{attribute 'linkalways'} 
{attribute 'no_explicit_call' := 'This FB is a CLASS and must be accessed using methods or properties'}
{attribute 'enable_dynamic_creation'}
FUNCTION_BLOCK _Array0to1OfUSINT EXTENDS ArrayDatatypeBase_1D
VAR CONSTANT
	lBound : DINT := 0;
	uBound : DINT := 1;
END_VAR
VAR
	localData : ARRAY [lBound..uBound] OF USINT;
	activeData : REFERENCE TO ARRAY [lBound..uBound] OF USINT REF= localData;
	elements : ARRAY [lBound..uBound] OF _USINT(0);
	baseType : _USINT(0);
END_VAR

PROPERTY PUBLIC Address : PVOID
GET
Address := ADR(activeData);
END_GET
END_PROPERTY

PROPERTY PUBLIC BaseDatatype : I_Datatype
GET
BaseDatatype := baseType;
END_GET
END_PROPERTY

METHOD PUBLIC ClearReference
VAR_INPUT
END_VAR
activeData REF= localData;
SetElementReference();
END_METHOD

METHOD PUBLIC Clone : I_Datatype
VAR
    pClone : POINTER TO _Array0to1OfUSINT;
END_VAR
pClone := __NEW(_Array0to1OfUSINT());
pClone^.Value := Value;
Clone := pClone^;
END_METHOD

METHOD FB_init : BOOL
VAR_INPUT
	bInitRetains : BOOL; // if TRUE, the retain variables are initialized (warm start / cold start)
	bInCopyCode : BOOL;  // if TRUE, the instance afterwards gets moved into the copy code (online change)
END_VAR
SetElementReference();
END_METHOD

METHOD PUBLIC MakeReferenceTo
VAR_INPUT
	ReferenceTarget : REFERENCE TO ARRAY [lBound..uBound] OF USINT;
END_VAR
activeData REF= ReferenceTarget;
SetElementReference();
END_METHOD

METHOD PROTECTED OnSerializeArrayValues
VAR_INPUT
	Serializer : I_Serializer;
END_VAR
VAR
	i : DINT;
END_VAR
FOR i := lBound TO uBound DO
	elements[i].SerializeWith(Serializer);
END_FOR
END_METHOD

METHOD PROTECTED SetElementReference
VAR_INPUT
END_VAR
VAR
	i : DINT;
END_VAR
FOR i := lBound TO uBound DO
	elements[i].MakeReferenceTo(activeData[i]);
END_FOR
END_METHOD

PROPERTY PUBLIC Size : UDINT
GET
Size := SIZEOF(activeData);
END_GET
END_PROPERTY

METHOD PROTECTED TryDeserializeArrayValues : BOOL
VAR_INPUT
	Deserializer : I_Deserializer;
	Feedback : I_DeserializerFeedback;
END_VAR
VAR
	enumerator : I_DeserializerArrayForwardEnumerator;
	i : DINT;
END_VAR
enumerator := Deserializer.GetArrayEnumerator();
i := lBound;

WHILE enumerator.MoveNext() AND i <= uBound DO
	
	IF NOT elements[i].TryDeserializeFrom(enumerator.Current, Feedback) THEN
		EXIT;
	END_IF
	i := i + 1;

END_WHILE
enumerator.Dispose();
END_METHOD

METHOD PUBLIC TryGetElementAsDatatypeByIndex : BOOL
VAR_INPUT
	Index : DINT;
	Destination : REFERENCE TO I_Datatype;
END_VAR
IF Index < lbound OR Index > ubound THEN
	RETURN;
END_IF

Destination := elements[Index];
TryGetElementAsDatatypeByIndex := TRUE;
END_METHOD

METHOD PUBLIC TryGetLowerBound : BOOL
VAR_INPUT
	Dimention : UDINT;
	Destination : REFERENCE TO DINT;
END_VAR
IF Dimention = 1 THEN
	Destination := lBound;
	TryGetLowerBound := TRUE;
END_IF
END_METHOD

METHOD PUBLIC TryGetUpperBound : BOOL
VAR_INPUT
	Dimention : UDINT;
	Destination : REFERENCE TO DINT;
END_VAR
IF Dimention = 1 THEN
	Destination := uBound;
	TryGetUpperBound := TRUE;
END_IF
END_METHOD

METHOD TryMakeReferenceTo : BOOL
VAR_INPUT
	Target : I_Datatype;
END_VAR
VAR
	pTargetData : POINTER TO ARRAY [lBound..uBound] OF USINT;
END_VAR
IF NOT IsEquivalentTo(Target) THEN
	RETURN;
END_IF

pTargetData := Target.Address;
activeData REF= pTargetData^;
SetElementReference();
TryMakeReferenceTo := TRUE;
END_METHOD

PROPERTY PUBLIC Value : REFERENCE TO ARRAY [lBound..uBound] OF USINT;
GET
Value ref= activeData;
END_GET
END_PROPERTY

END_FUNCTION_BLOCK

(* stored: Version 1.1.0.1, ProductVersion 3.1.4024.13
   POU _Array0to1OfUSINT: Id {809f4d15-75a6-0d4d-342f-d4df08bef26b}, SpecialFunc None
   Folder Core: Id {20405364-43c1-0360-3f13-c7b6b46347e7}
   Folder Constructor: Id {908c995d-d65e-0f17-2c61-dd1428a238a9}
   Folder Protected: Id {dfab63e4-fcbe-0bc7-0ff3-1ff4a2700262}
   Folder Customize: Id {9282016e-9e25-0a51-3ea2-b0f729feb462}
   Property Address: Id {ad213f99-3e13-0541-3bbf-09cab285d405}
   Get Get: Id {3ed5b802-24ab-0f0e-0445-8231e37b8cbd}
   Property BaseDatatype: Id {7ef03571-8bc5-0247-333b-5691cc5bf9a1}
   Get Get: Id {de10912a-e5a7-03eb-05d8-57eb7747a96a}
   Method ClearReference: Id {ce4594e1-2b13-0cda-2807-59ba5d9189e5}
   Method Clone: Id {64423a02-b6d0-0e8a-0760-8bfc10b30d4b}
   Method FB_init: Id {406c2806-71c0-00af-1989-a14c1a329468}
   Method MakeReferenceTo: Id {5b4f1f2e-542e-0474-1042-eaa2ddcf0ffe}
   Method OnSerializeArrayValues: Id {b21bb398-199d-0e16-31a8-cd09df871397}
   Method SetElementReference: Id {7c9dd691-accb-0531-2dc9-c10ab7ee6fcb}
   Property Size: Id {49787b77-9a41-0c14-15da-d9010493de80}
   Get Get: Id {5634b85b-70c4-0de8-2a44-a0a05d06768a}
   Method TryDeserializeArrayValues: Id {02d736b4-f63d-0bf4-14f9-cfb9fc342882}
   Method TryGetElementAsDatatypeByIndex: Id {32fcd423-74eb-05b7-378c-6b6a234ace87}
   Method TryGetLowerBound: Id {cbf098bf-2dc2-04a7-3516-030d4bd95e11}
   Method TryGetUpperBound: Id {6d144c83-c8ac-0241-2669-af811d77153e}
   Method TryMakeReferenceTo: Id {35d6b41d-26dc-0da1-3296-f9118f52badc}
   Property Value: Id {9fd1d8b9-666f-0267-1093-36a856a86a1e}
   Get Get: Id {08683395-9af3-0833-1de8-802a8bf4e718} *)
